// TIA Portal project "ap2s71200exam_V15.1" (V15.1)

(* hardware
DEVICE "S7-1200 station_1"  S7-1200 Station
   slot 0: "Rack_0"  S7-1200 Rack  Rack  V1.0
   slot 1: "PLC_1"  CPU 1214C DC/DC/DC  6ES7 214-1AG40-0XB0  V4.2
   slot 2: "DI 16/DQ 16x24VDC_1"  6ES7 223-1BL32-0XB0  V2.0
*)

// ===== PLC "PLC_1"  CPU 1214C DC/DC/DC =====

VAR_GLOBAL   // PLC tag table "Default tag table"
   "-F5" AT %I0.0 : Bool;
   "-S3" AT %I0.1 : Bool;
   "-S4" AT %I0.2 : Bool;
   "-S5" AT %I0.3 : Bool;
   "-S6" AT %I0.4 : Bool;
   "-S7" AT %I0.5 : Bool;
   "-S8" AT %I0.6 : Bool;
   "-S9" AT %I0.7 : Bool;
   "-S10" AT %I1.0 : Bool;
   "-S11" AT %I1.1 : Bool;
   "-S12" AT %I1.2 : Bool;
   "-BP1" AT %I1.3 : Bool;
   "-B11" AT %I1.4 : Bool;
   "-B12" AT %I1.5 : Bool;
   "-B13" AT %I2.0 : Bool;
   "-B21" AT %I2.1 : Bool;
   "-B22" AT %I2.2 : Bool;
   "-B31" AT %I2.3 : Bool;
   "-B32" AT %I2.4 : Bool;
   "-B53" AT %I2.5 : Bool;
   "Reserve2" AT %I2.6 : Bool;
   "Reserve3" AT %I2.7 : Bool;
   "-B52" AT %I3.0 : Bool;
   "-F7" AT %I3.1 : Bool;
   "-M21" AT %Q0.0 : Bool;
   "-M22" AT %Q0.1 : Bool;
   "-M31" AT %Q0.2 : Bool;
   "-M32" AT %Q0.3 : Bool;
   "Reserve5" AT %Q0.4 : Bool;
   "Reserve6" AT %Q0.5 : Bool;
   "-Q5" AT %Q0.6 : Bool;
   "-Q6" AT %Q0.7 : Bool;
   "-P32" AT %Q2.0 : Bool;
   "Reserve7" AT %Q2.1 : Bool;
   "-Q60" AT %Q2.2 : Bool;
   "-P2" AT %Q2.3 : Bool;
   "-P3" AT %Q2.4 : Bool;
   "-P4" AT %Q2.5 : Bool;
   "-P5" AT %Q2.6 : Bool;
   "-P6" AT %Q2.7 : Bool;
   "-P7" AT %Q3.0 : Bool;
   "-P8" AT %Q3.1 : Bool;
   "-P10" AT %Q3.2 : Bool;
   "-P11" AT %Q3.3 : Bool;
   "-P12" AT %Q3.4 : Bool;
   "-P13" AT %Q3.5 : Bool;
   "-P14" AT %Q3.6 : Bool;
   "-Reserve8" AT %Q3.7 : Bool;
END_VAR

DATA_BLOCK "G_Master_DB"   // DB12
{ S7_Optimized_Access := 'TRUE' }
VERSION : 0.1
// stored: InstanceOfName G_Master
"G_Master"
BEGIN
END_DATA_BLOCK

DATA_BLOCK "G_Clock_DB"   // DB13
{ S7_Optimized_Access := 'TRUE' }
VERSION : 0.1
// stored: InstanceOfName G_Clock
"G_Clock"
BEGIN
END_DATA_BLOCK

DATA_BLOCK "G_Indicator_DB"   // DB14
{ S7_Optimized_Access := 'TRUE' }
VERSION : 0.1
// stored: InstanceOfName G_Indicator
"G_Indicator"
BEGIN
END_DATA_BLOCK

DATA_BLOCK "G_Settings_DB"   // DB15
{ S7_Optimized_Access := 'TRUE' }
VERSION : 0.1
// stored: InstanceOfName G_Settings
"G_Settings"
BEGIN
END_DATA_BLOCK

DATA_BLOCK "G_Autos_DB"   // DB16
{ S7_Optimized_Access := 'TRUE' }
VERSION : 0.1
// stored: InstanceOfName G_Autos
"G_Autos"
BEGIN
END_DATA_BLOCK

DATA_BLOCK "Output total_DB"   // DB17
{ S7_Optimized_Access := 'TRUE' }
VERSION : 0.1
// stored: InstanceOfName Output total
"Output total"
BEGIN
END_DATA_BLOCK

// folder: System blocks/Program resources

DATA_BLOCK "0.5s/G_Clock.X100"   // DB1
{ S7_Optimized_Access := 'TRUE' }
AUTHOR : Simatic
FAMILY : IEC
NAME : IEC_TMR
VERSION : 1.0
// stored: InstanceOfName IEC_TIMER
"IEC_TIMER"
BEGIN
END_DATA_BLOCK

DATA_BLOCK "0.5s/G_Clock.X101"   // DB2
{ S7_Optimized_Access := 'TRUE' }
AUTHOR : Simatic
FAMILY : IEC
NAME : IEC_TMR
VERSION : 1.0
// stored: InstanceOfName IEC_TIMER
"IEC_TIMER"
BEGIN
END_DATA_BLOCK

DATA_BLOCK "1s/B11.X501"   // DB3
{ S7_Optimized_Access := 'TRUE' }
AUTHOR : Simatic
FAMILY : IEC
NAME : IEC_TMR
VERSION : 1.0
// stored: InstanceOfName IEC_TIMER
"IEC_TIMER"
BEGIN
END_DATA_BLOCK

DATA_BLOCK "1s/B22.X502"   // DB4
{ S7_Optimized_Access := 'TRUE' }
AUTHOR : Simatic
FAMILY : IEC
NAME : IEC_TMR
VERSION : 1.0
// stored: InstanceOfName IEC_TIMER
"IEC_TIMER"
BEGIN
END_DATA_BLOCK

DATA_BLOCK "1s/B21.X503"   // DB5
{ S7_Optimized_Access := 'TRUE' }
AUTHOR : Simatic
FAMILY : IEC
NAME : IEC_TMR
VERSION : 1.0
// stored: InstanceOfName IEC_TIMER
"IEC_TIMER"
BEGIN
END_DATA_BLOCK

DATA_BLOCK "1s/B13.X504"   // DB6
{ S7_Optimized_Access := 'TRUE' }
AUTHOR : Simatic
FAMILY : IEC
NAME : IEC_TMR
VERSION : 1.0
// stored: InstanceOfName IEC_TIMER
"IEC_TIMER"
BEGIN
END_DATA_BLOCK

DATA_BLOCK "1s/B22.X505"   // DB7
{ S7_Optimized_Access := 'TRUE' }
AUTHOR : Simatic
FAMILY : IEC
NAME : IEC_TMR
VERSION : 1.0
// stored: InstanceOfName IEC_TIMER
"IEC_TIMER"
BEGIN
END_DATA_BLOCK

DATA_BLOCK "1s/Q60.X506"   // DB8
{ S7_Optimized_Access := 'TRUE' }
AUTHOR : Simatic
FAMILY : IEC
NAME : IEC_TMR
VERSION : 1.0
// stored: InstanceOfName IEC_TIMER
"IEC_TIMER"
BEGIN
END_DATA_BLOCK

DATA_BLOCK "1s/B21.X507"   // DB9
{ S7_Optimized_Access := 'TRUE' }
AUTHOR : Simatic
FAMILY : IEC
NAME : IEC_TMR
VERSION : 1.0
// stored: InstanceOfName IEC_TIMER
"IEC_TIMER"
BEGIN
END_DATA_BLOCK

DATA_BLOCK "1s/B32.X508"   // DB10
{ S7_Optimized_Access := 'TRUE' }
AUTHOR : Simatic
FAMILY : IEC
NAME : IEC_TMR
VERSION : 1.0
// stored: InstanceOfName IEC_TIMER
"IEC_TIMER"
BEGIN
END_DATA_BLOCK

DATA_BLOCK "1s/B31.X509"   // DB11
{ S7_Optimized_Access := 'TRUE' }
AUTHOR : Simatic
FAMILY : IEC
NAME : IEC_TMR
VERSION : 1.0
// stored: InstanceOfName IEC_TIMER
"IEC_TIMER"
BEGIN
END_DATA_BLOCK

// folder: (top level)

FUNCTION_BLOCK "G_Master"   // FB1, FBD
{ S7_Optimized_Access := 'TRUE' }
VERSION : 0.1
   VAR_INPUT
      F5 : Bool;
      F7 : Bool;
      BP1 : Bool;
      S3 : Bool;
      S4 : Bool;
      "1Hz" : Bool;
      "G_setting.X300" : Bool;
      "G_auto.X500" : Bool;
   END_VAR
   VAR_OUTPUT
      G_setting : Bool;
      G_auto : Bool;
      P3 : Bool;
   END_VAR
   VAR
      X1 : Bool;
      X2 : Bool;
      X3 : Bool;
      X4 : Bool;
      X5 : Bool;
   END_VAR
BEGIN

REGION Network 1
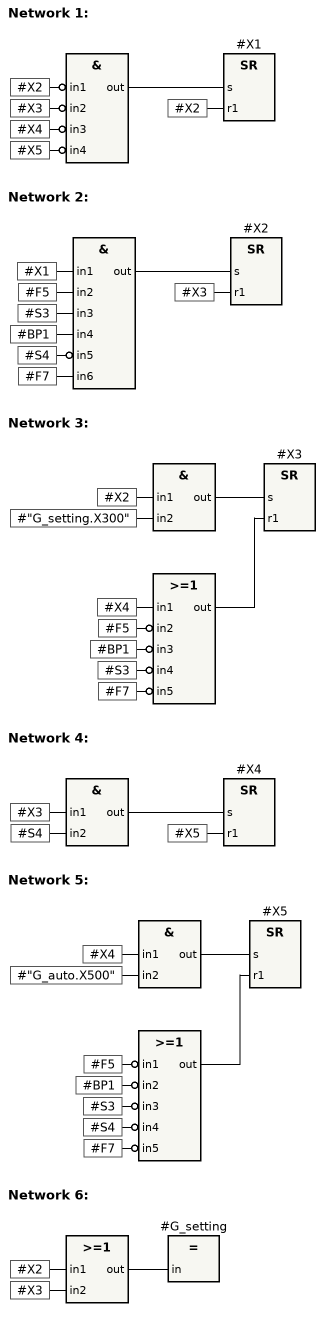
   IF NOT #X2 AND NOT #X3 AND NOT #X4 AND NOT #X5 THEN
       #X1 := TRUE;   // SR flip-flop
   END_IF;
   IF #X2 THEN #X1 := FALSE; END_IF;
END_REGION

REGION Network 2
   IF #X1 AND #F5 AND #S3 AND #BP1 AND NOT #S4 AND #F7 THEN
       #X2 := TRUE;   // SR flip-flop
   END_IF;
   IF #X3 THEN #X2 := FALSE; END_IF;
END_REGION

REGION Network 3
   IF #X2 AND #"G_setting.X300" THEN
       #X3 := TRUE;   // SR flip-flop
   END_IF;
   IF #X4 OR NOT #F5 OR NOT #BP1 OR NOT #S3 OR NOT #F7 THEN #X3 := FALSE; END_IF;
END_REGION

REGION Network 4
   IF #X3 AND #S4 THEN
       #X4 := TRUE;   // SR flip-flop
   END_IF;
   IF #X5 THEN #X4 := FALSE; END_IF;
END_REGION

REGION Network 5
   IF #X4 AND #"G_auto.X500" THEN
       #X5 := TRUE;   // SR flip-flop
   END_IF;
   IF NOT #F5 OR NOT #BP1 OR NOT #S3 OR NOT #S4 OR NOT #F7 THEN #X5 := FALSE; END_IF;
END_REGION

REGION Network 6
   #G_setting := #X2 OR #X3;
END_REGION

REGION Network 7
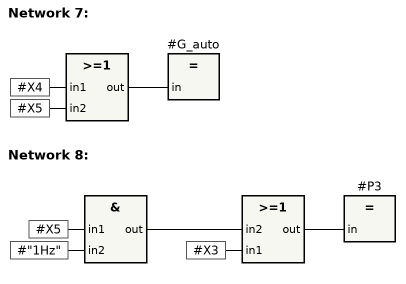
   #G_auto := #X4 OR #X5;
END_REGION

REGION Network 8
   #P3 := (#X5 AND #"1Hz") OR #X3;
END_REGION
END_FUNCTION_BLOCK

FUNCTION_BLOCK "G_Clock"   // FB2, FBD
{ S7_Optimized_Access := 'TRUE' }
VERSION : 0.1
   VAR_OUTPUT
      "1Hz" : Bool;
   END_VAR
   VAR
      X100 : Bool;
      X101 : Bool;
   END_VAR
BEGIN

REGION Network 1
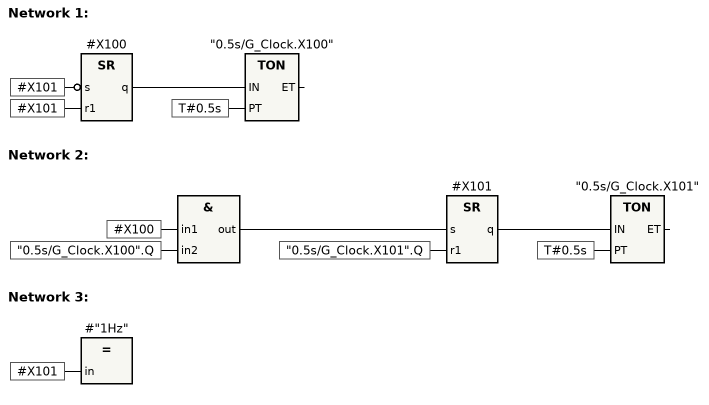
   IF NOT #X101 THEN
       #X100 := TRUE;   // SR flip-flop
   END_IF;
   IF #X101 THEN #X100 := FALSE; END_IF;
   "0.5s/G_Clock.X100".TON(IN := #X100, PT := T#0.5s);
END_REGION

REGION Network 2
   IF #X100 AND "0.5s/G_Clock.X100".Q THEN
       #X101 := TRUE;   // SR flip-flop
   END_IF;
   IF "0.5s/G_Clock.X101".Q THEN #X101 := FALSE; END_IF;
   "0.5s/G_Clock.X101".TON(IN := #X101, PT := T#0.5s);
END_REGION

REGION Network 3
   #"1Hz" := #X101;
END_REGION
END_FUNCTION_BLOCK

FUNCTION_BLOCK "G_Indicator"   // FB3, FBD
{ S7_Optimized_Access := 'TRUE' }
VERSION : 0.1
   VAR_INPUT
      S3 : Bool;
      S4 : Bool;
      F7 : Bool;
      "1Hz" : Bool;
      BP1 : Bool;
      B11 : Bool;
      B12 : Bool;
      B13 : Bool;
      B21 : Bool;
      B22 : Bool;
      B31 : Bool;
      B32 : Bool;
      B52 : Bool;
      B53 : Bool;
      Q5_In : Bool;
      Q6_In : Bool;
      Q60_In : Bool;
   END_VAR
   VAR_OUTPUT
      P2 : Bool;
      P3 : Bool;
      P4 : Bool;
      P5 : Bool;
      P6 : Bool;
      P7 : Bool;
      P8 : Bool;
      P10 : Bool;
      P11 : Bool;
      P12 : Bool;
      P13 : Bool;
      P14 : Bool;
      P32 : Bool;
   END_VAR
   VAR
      X200 : Bool;
      X201 : Bool;
   END_VAR
BEGIN

REGION Network 1
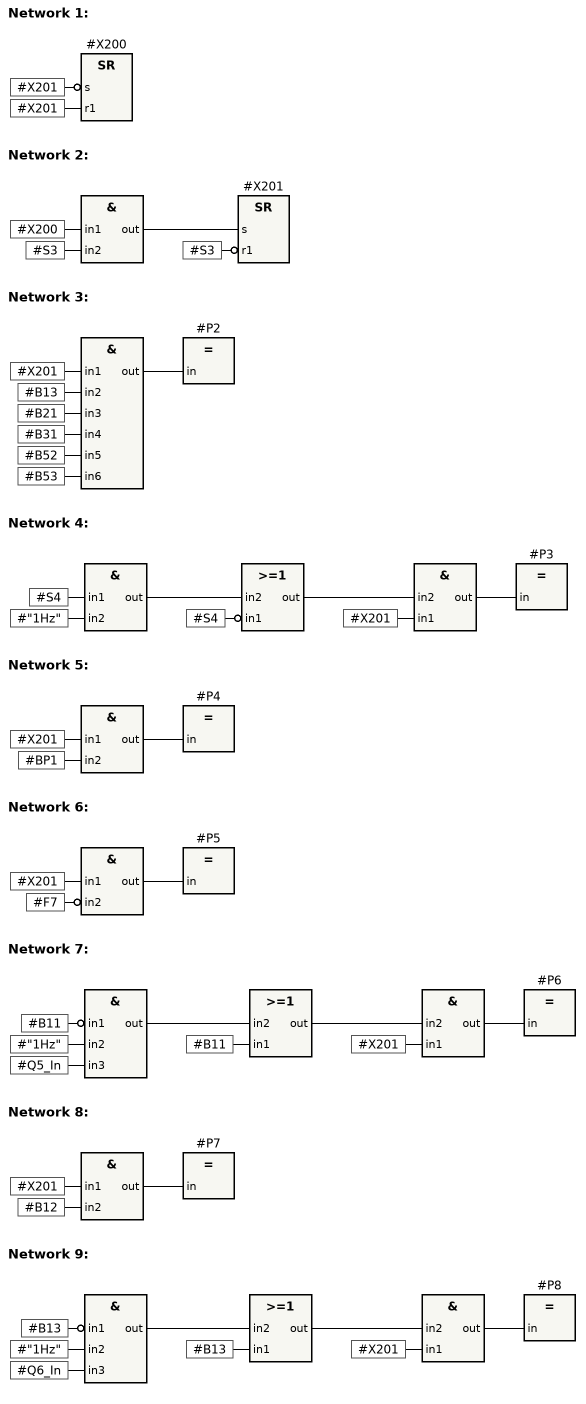
   IF NOT #X201 THEN
       #X200 := TRUE;   // SR flip-flop
   END_IF;
   IF #X201 THEN #X200 := FALSE; END_IF;
END_REGION

REGION Network 2
   IF #X200 AND #S3 THEN
       #X201 := TRUE;   // SR flip-flop
   END_IF;
   IF NOT #S3 THEN #X201 := FALSE; END_IF;
END_REGION

REGION Network 3
   #P2 := #X201 AND #B13 AND #B21 AND #B31 AND #B52 AND #B53;
END_REGION

REGION Network 4
   #P3 := ((#S4 AND #"1Hz") OR NOT #S4) AND #X201;
END_REGION

REGION Network 5
   #P4 := #X201 AND #BP1;
END_REGION

REGION Network 6
   #P5 := #X201 AND NOT #F7;
END_REGION

REGION Network 7
   #P6 := ((NOT #B11 AND #"1Hz" AND #Q5_In) OR #B11) AND #X201;
END_REGION

REGION Network 8
   #P7 := #X201 AND #B12;
END_REGION

REGION Network 9
   #P8 := ((NOT #B13 AND #"1Hz" AND #Q6_In) OR #B13) AND #X201;
END_REGION

REGION Network 10
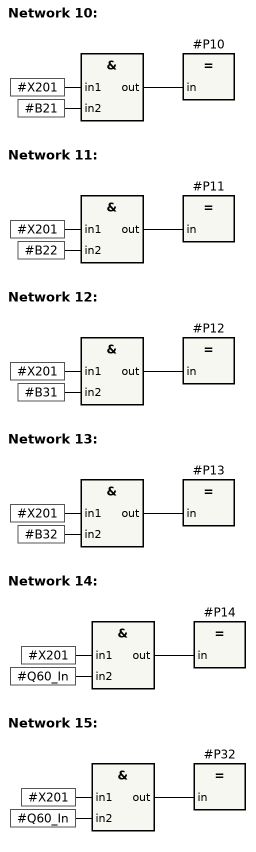
   #P10 := #X201 AND #B21;
END_REGION

REGION Network 11
   #P11 := #X201 AND #B22;
END_REGION

REGION Network 12
   #P12 := #X201 AND #B31;
END_REGION

REGION Network 13
   #P13 := #X201 AND #B32;
END_REGION

REGION Network 14
   #P14 := #X201 AND #Q60_In;
END_REGION

REGION Network 15
   #P32 := #X201 AND #Q60_In;
END_REGION
END_FUNCTION_BLOCK

FUNCTION_BLOCK "G_Settings"   // FB4, FBD
{ S7_Optimized_Access := 'TRUE' }
VERSION : 0.1
   VAR_INPUT
      G_setting : Bool;
      S4 : Bool;
      S6 : Bool;
      S7 : Bool;
      S8 : Bool;
      S9 : Bool;
      S10 : Bool;
      S11 : Bool;
      S12 : Bool;
      B11 : Bool;
      B13 : Bool;
      B21 : Bool;
   END_VAR
   VAR_OUTPUT
      Q5_S : Bool;
      Q6_S : Bool;
      Q60_S : Bool;
      M21_S : Bool;
      M22_S : Bool;
      M31_S : Bool;
      M32_S : Bool;
   END_VAR
   VAR
      X300 : Bool;
      X301 : Bool;
   END_VAR
BEGIN

REGION Network 1
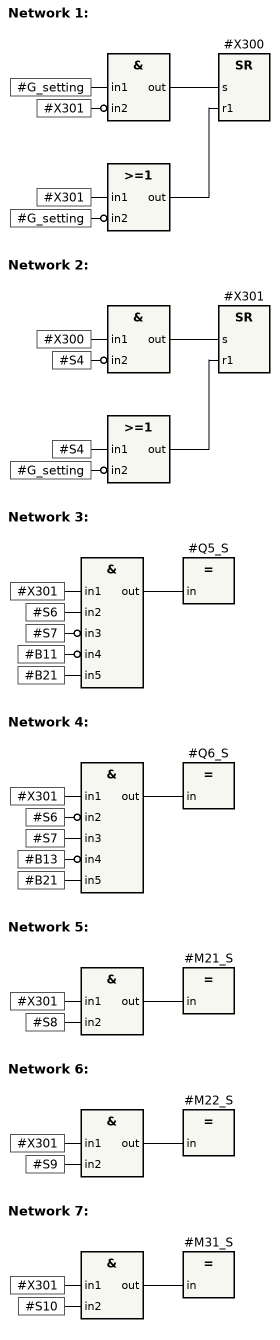
   IF #G_setting AND NOT #X301 THEN
       #X300 := TRUE;   // SR flip-flop
   END_IF;
   IF #X301 OR NOT #G_setting THEN #X300 := FALSE; END_IF;
END_REGION

REGION Network 2
   IF #X300 AND NOT #S4 THEN
       #X301 := TRUE;   // SR flip-flop
   END_IF;
   IF #S4 OR NOT #G_setting THEN #X301 := FALSE; END_IF;
END_REGION

REGION Network 3
   #Q5_S := #X301 AND #S6 AND NOT #S7 AND NOT #B11 AND #B21;
END_REGION

REGION Network 4
   #Q6_S := #X301 AND NOT #S6 AND #S7 AND NOT #B13 AND #B21;
END_REGION

REGION Network 5
   #M21_S := #X301 AND #S8;
END_REGION

REGION Network 6
   #M22_S := #X301 AND #S9;
END_REGION

REGION Network 7
   #M31_S := #X301 AND #S10;
END_REGION

REGION Network 8
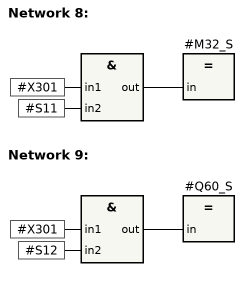
   #M32_S := #X301 AND #S11;
END_REGION

REGION Network 9
   #Q60_S := #X301 AND #S12;
END_REGION
END_FUNCTION_BLOCK

FUNCTION_BLOCK "G_Autos"   // FB5, FBD
{ S7_Optimized_Access := 'TRUE' }
VERSION : 0.1
   VAR_INPUT
      G_auto : Bool;
      S5 : Bool;
      B11 : Bool;
      B12 : Bool;
      B13 : Bool;
      B21 : Bool;
      B22 : Bool;
      B31 : Bool;
      B32 : Bool;
      B52 : Bool;
      B53 : Bool;
      Q60_In : Bool;
   END_VAR
   VAR_OUTPUT
      Q5_A : Bool;
      Q6_A : Bool;
      Q60_A : Bool;
      M21_A : Bool;
      M22_A : Bool;
      M31_A : Bool;
      M32_A : Bool;
   END_VAR
   VAR
      X500 : Bool;
      X501 : Bool;
      X502 : Bool;
      X503 : Bool;
      X504 : Bool;
      X505 : Bool;
      X506 : Bool;
      X507 : Bool;
      X508 : Bool;
      X509 : Bool;
   END_VAR
BEGIN

REGION Network 1
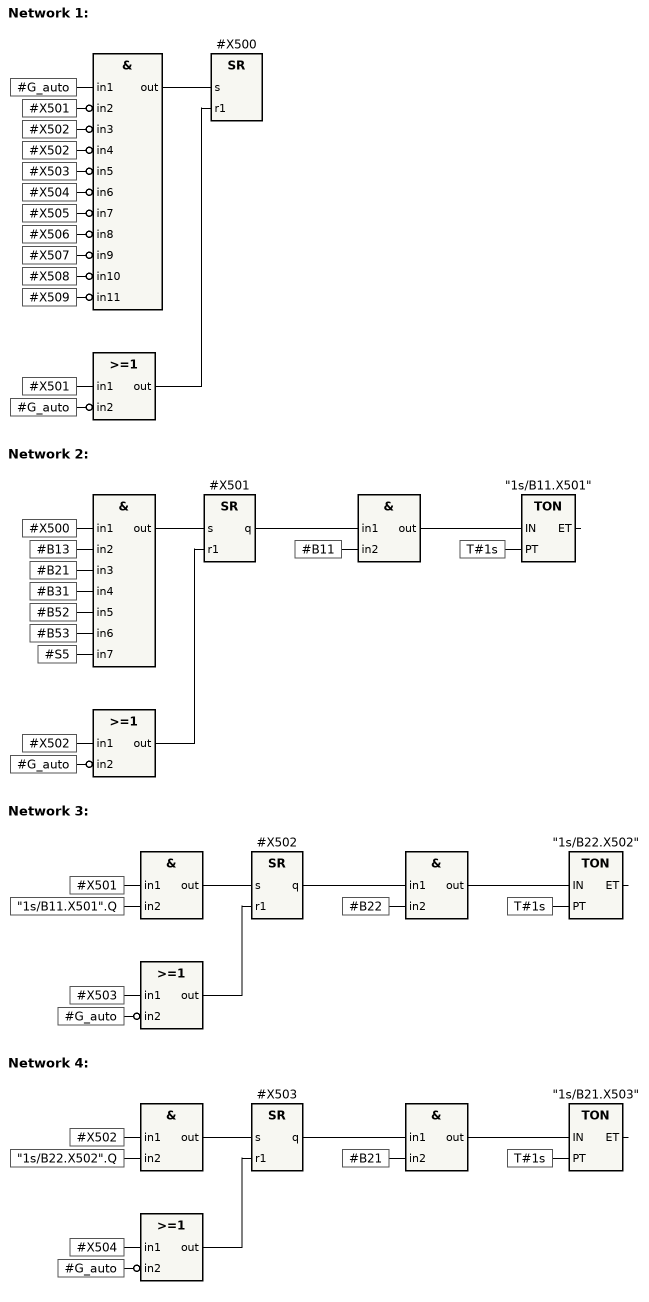
   IF #G_auto AND NOT #X501 AND NOT #X502 AND NOT #X502 AND NOT #X503 AND NOT #X504 AND NOT #X505 AND NOT #X506 AND NOT #X507 AND NOT #X508 AND NOT #X509 THEN
       #X500 := TRUE;   // SR flip-flop
   END_IF;
   IF #X501 OR NOT #G_auto THEN #X500 := FALSE; END_IF;
END_REGION

REGION Network 2
   IF #X500 AND #B13 AND #B21 AND #B31 AND #B52 AND #B53 AND #S5 THEN
       #X501 := TRUE;   // SR flip-flop
   END_IF;
   IF #X502 OR NOT #G_auto THEN #X501 := FALSE; END_IF;
   "1s/B11.X501".TON(IN := #X501 AND #B11, PT := T#1s);
END_REGION

REGION Network 3
   IF #X501 AND "1s/B11.X501".Q THEN
       #X502 := TRUE;   // SR flip-flop
   END_IF;
   IF #X503 OR NOT #G_auto THEN #X502 := FALSE; END_IF;
   "1s/B22.X502".TON(IN := #X502 AND #B22, PT := T#1s);
END_REGION

REGION Network 4
   IF #X502 AND "1s/B22.X502".Q THEN
       #X503 := TRUE;   // SR flip-flop
   END_IF;
   IF #X504 OR NOT #G_auto THEN #X503 := FALSE; END_IF;
   "1s/B21.X503".TON(IN := #X503 AND #B21, PT := T#1s);
END_REGION

REGION Network 5
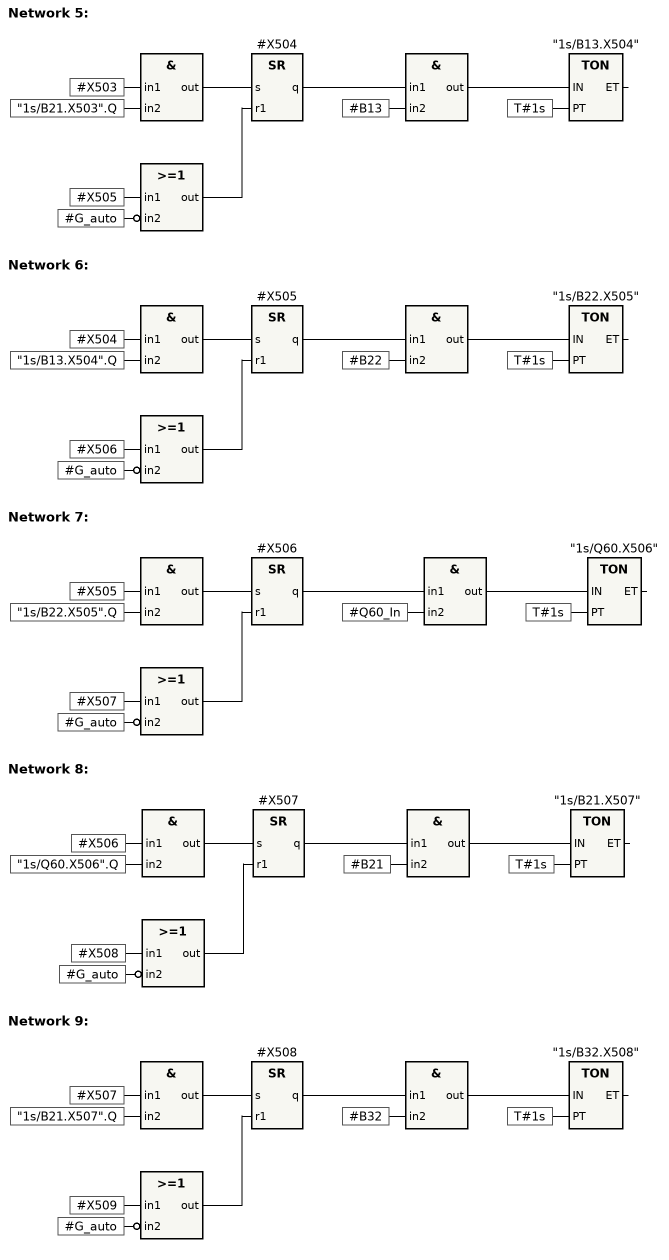
   IF #X503 AND "1s/B21.X503".Q THEN
       #X504 := TRUE;   // SR flip-flop
   END_IF;
   IF #X505 OR NOT #G_auto THEN #X504 := FALSE; END_IF;
   "1s/B13.X504".TON(IN := #X504 AND #B13, PT := T#1s);
END_REGION

REGION Network 6
   IF #X504 AND "1s/B13.X504".Q THEN
       #X505 := TRUE;   // SR flip-flop
   END_IF;
   IF #X506 OR NOT #G_auto THEN #X505 := FALSE; END_IF;
   "1s/B22.X505".TON(IN := #X505 AND #B22, PT := T#1s);
END_REGION

REGION Network 7
   IF #X505 AND "1s/B22.X505".Q THEN
       #X506 := TRUE;   // SR flip-flop
   END_IF;
   IF #X507 OR NOT #G_auto THEN #X506 := FALSE; END_IF;
   "1s/Q60.X506".TON(IN := #X506 AND #Q60_In, PT := T#1s);
END_REGION

REGION Network 8
   IF #X506 AND "1s/Q60.X506".Q THEN
       #X507 := TRUE;   // SR flip-flop
   END_IF;
   IF #X508 OR NOT #G_auto THEN #X507 := FALSE; END_IF;
   "1s/B21.X507".TON(IN := #X507 AND #B21, PT := T#1s);
END_REGION

REGION Network 9
   IF #X507 AND "1s/B21.X507".Q THEN
       #X508 := TRUE;   // SR flip-flop
   END_IF;
   IF #X509 OR NOT #G_auto THEN #X508 := FALSE; END_IF;
   "1s/B32.X508".TON(IN := #X508 AND #B32, PT := T#1s);
END_REGION

REGION Network 10
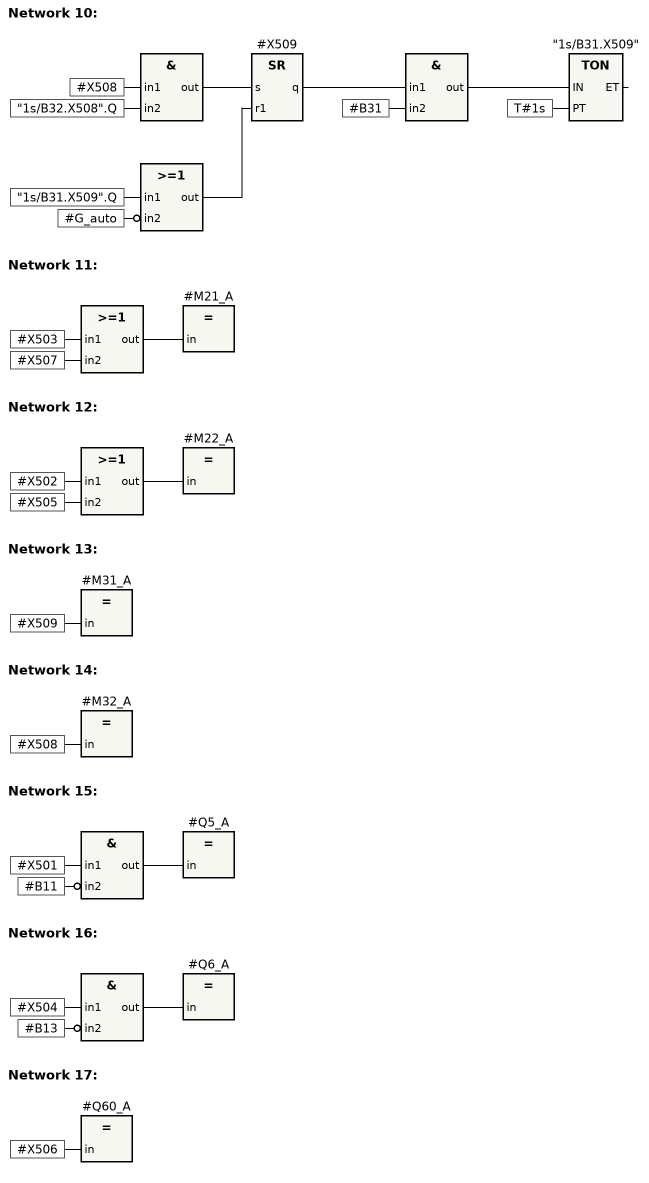
   IF #X508 AND "1s/B32.X508".Q THEN
       #X509 := TRUE;   // SR flip-flop
   END_IF;
   IF "1s/B31.X509".Q OR NOT #G_auto THEN #X509 := FALSE; END_IF;
   "1s/B31.X509".TON(IN := #X509 AND #B31, PT := T#1s);
END_REGION

REGION Network 11
   #M21_A := #X503 OR #X507;
END_REGION

REGION Network 12
   #M22_A := #X502 OR #X505;
END_REGION

REGION Network 13
   #M31_A := #X509;
END_REGION

REGION Network 14
   #M32_A := #X508;
END_REGION

REGION Network 15
   #Q5_A := #X501 AND NOT #B11;
END_REGION

REGION Network 16
   #Q6_A := #X504 AND NOT #B13;
END_REGION

REGION Network 17
   #Q60_A := #X506;
END_REGION
END_FUNCTION_BLOCK

FUNCTION_BLOCK "Output total"   // FB6, FBD
{ S7_Optimized_Access := 'TRUE' }
VERSION : 0.1
   VAR_INPUT
      M21_A : Bool;
      M22_A : Bool;
      M31_A : Bool;
      M32_A : Bool;
      Q5_A : Bool;
      Q6_A : Bool;
      Q60_A : Bool;
      M21_S : Bool;
      M22_S : Bool;
      M31_S : Bool;
      M32_S : Bool;
      Q5_S : Bool;
      Q6_S : Bool;
      Q60_S : Bool;
   END_VAR
   VAR_OUTPUT
      M21 : Bool;
      M22 : Bool;
      M31 : Bool;
      M32 : Bool;
      Q5 : Bool;
      Q6 : Bool;
      Q60 : Bool;
   END_VAR
BEGIN

REGION Network 1
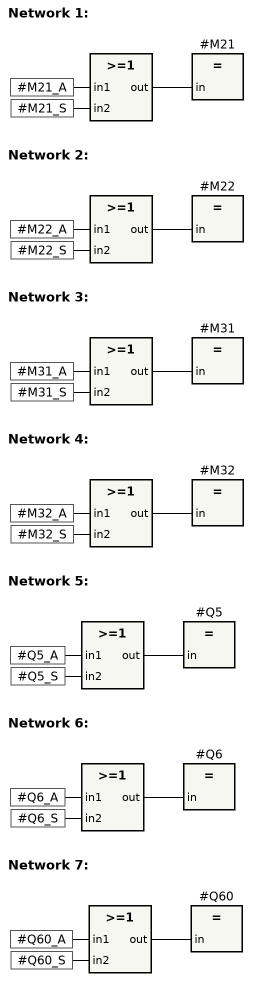
   #M21 := #M21_A OR #M21_S;
END_REGION

REGION Network 2
   #M22 := #M22_A OR #M22_S;
END_REGION

REGION Network 3
   #M31 := #M31_A OR #M31_S;
END_REGION

REGION Network 4
   #M32 := #M32_A OR #M32_S;
END_REGION

REGION Network 5
   #Q5 := #Q5_A OR #Q5_S;
END_REGION

REGION Network 6
   #Q6 := #Q6_A OR #Q6_S;
END_REGION

REGION Network 7
   #Q60 := #Q60_A OR #Q60_S;
END_REGION
END_FUNCTION_BLOCK

ORGANIZATION_BLOCK "Main"   // OB1, FBD, ProgramCycle
TITLE = "Main Program Sweep (Cycle)"
{ S7_Optimized_Access := 'TRUE' }
VERSION : 0.1
   VAR_INPUT
      Initial_Call : Bool;   // Initial call of this OB
      Remanence : Bool;   // =True, if remanent data are available
   END_VAR
BEGIN

REGION Network 1
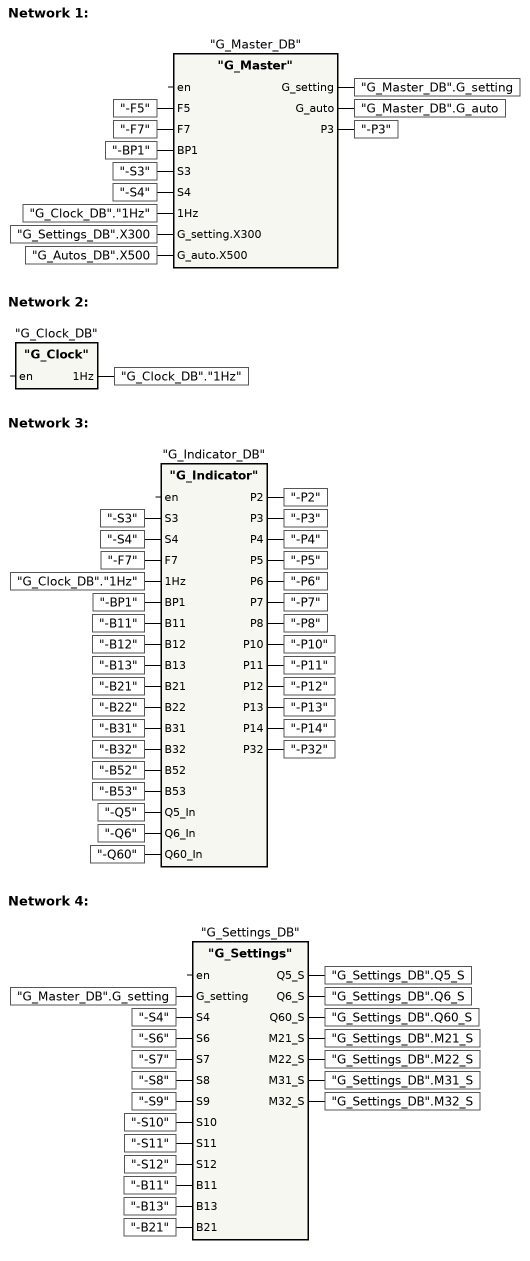
   "G_Master_DB"(F5 := "-F5",   // "G_Master"
                 F7 := "-F7",
                 BP1 := "-BP1",
                 S3 := "-S3",
                 S4 := "-S4",
                 "1Hz" := "G_Clock_DB"."1Hz",
                 "G_setting.X300" := "G_Settings_DB".X300,
                 "G_auto.X500" := "G_Autos_DB".X500,
                 G_setting => "G_Master_DB".G_setting,
                 G_auto => "G_Master_DB".G_auto,
                 P3 => "-P3");
END_REGION

REGION Network 2
   "G_Clock_DB"("1Hz" => "G_Clock_DB"."1Hz");   // "G_Clock"
END_REGION

REGION Network 3
   "G_Indicator_DB"(S3 := "-S3",   // "G_Indicator"
                    S4 := "-S4",
                    F7 := "-F7",
                    "1Hz" := "G_Clock_DB"."1Hz",
                    BP1 := "-BP1",
                    B11 := "-B11",
                    B12 := "-B12",
                    B13 := "-B13",
                    B21 := "-B21",
                    B22 := "-B22",
                    B31 := "-B31",
                    B32 := "-B32",
                    B52 := "-B52",
                    B53 := "-B53",
                    Q5_In := "-Q5",
                    Q6_In := "-Q6",
                    Q60_In := "-Q60",
                    P2 => "-P2",
                    P3 => "-P3",
                    P4 => "-P4",
                    P5 => "-P5",
                    P6 => "-P6",
                    P7 => "-P7",
                    P8 => "-P8",
                    P10 => "-P10",
                    P11 => "-P11",
                    P12 => "-P12",
                    P13 => "-P13",
                    P14 => "-P14",
                    P32 => "-P32");
END_REGION

REGION Network 4
   "G_Settings_DB"(G_setting := "G_Master_DB".G_setting,   // "G_Settings"
                   S4 := "-S4",
                   S6 := "-S6",
                   S7 := "-S7",
                   S8 := "-S8",
                   S9 := "-S9",
                   S10 := "-S10",
                   S11 := "-S11",
                   S12 := "-S12",
                   B11 := "-B11",
                   B13 := "-B13",
                   B21 := "-B21",
                   Q5_S => "G_Settings_DB".Q5_S,
                   Q6_S => "G_Settings_DB".Q6_S,
                   Q60_S => "G_Settings_DB".Q60_S,
                   M21_S => "G_Settings_DB".M21_S,
                   M22_S => "G_Settings_DB".M22_S,
                   M31_S => "G_Settings_DB".M31_S,
                   M32_S => "G_Settings_DB".M32_S);
END_REGION

REGION Network 5
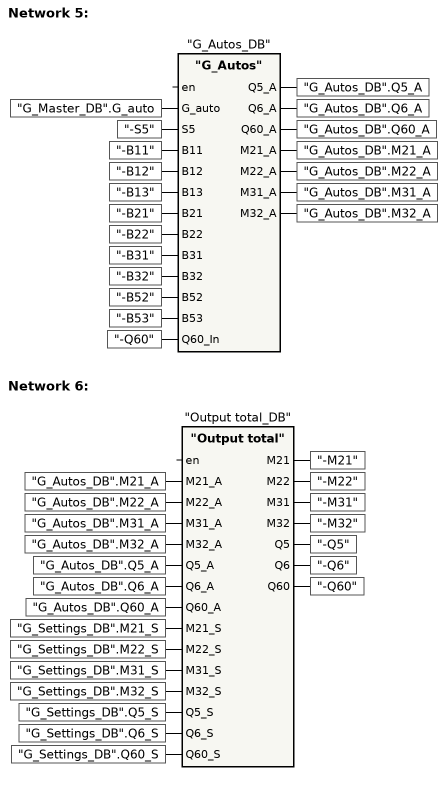
   "G_Autos_DB"(G_auto := "G_Master_DB".G_auto,   // "G_Autos"
                S5 := "-S5",
                B11 := "-B11",
                B12 := "-B12",
                B13 := "-B13",
                B21 := "-B21",
                B22 := "-B22",
                B31 := "-B31",
                B32 := "-B32",
                B52 := "-B52",
                B53 := "-B53",
                Q60_In := "-Q60",
                Q5_A => "G_Autos_DB".Q5_A,
                Q6_A => "G_Autos_DB".Q6_A,
                Q60_A => "G_Autos_DB".Q60_A,
                M21_A => "G_Autos_DB".M21_A,
                M22_A => "G_Autos_DB".M22_A,
                M31_A => "G_Autos_DB".M31_A,
                M32_A => "G_Autos_DB".M32_A);
END_REGION

REGION Network 6
   "Output total_DB"(M21_A := "G_Autos_DB".M21_A,   // "Output total"
                     M22_A := "G_Autos_DB".M22_A,
                     M31_A := "G_Autos_DB".M31_A,
                     M32_A := "G_Autos_DB".M32_A,
                     Q5_A := "G_Autos_DB".Q5_A,
                     Q6_A := "G_Autos_DB".Q6_A,
                     Q60_A := "G_Autos_DB".Q60_A,
                     M21_S := "G_Settings_DB".M21_S,
                     M22_S := "G_Settings_DB".M22_S,
                     M31_S := "G_Settings_DB".M31_S,
                     M32_S := "G_Settings_DB".M32_S,
                     Q5_S := "G_Settings_DB".Q5_S,
                     Q6_S := "G_Settings_DB".Q6_S,
                     Q60_S := "G_Settings_DB".Q60_S,
                     M21 => "-M21",
                     M22 => "-M22",
                     M31 => "-M31",
                     M32 => "-M32",
                     Q5 => "-Q5",
                     Q6 => "-Q6",
                     Q60 => "-Q60");
END_REGION
END_ORGANIZATION_BLOCK